// TIA Portal V17 export
// export: Created 2022-12-09T10:51:17.2356961Z, ExportSetting WithDefaults, DisplayName Totally Integrated Automation Portal, DisplayVersion V17 Update 5, DisplayName TIA Portal Openness, DisplayVersion V17 Update 5, DisplayName TIA Portal Version Control Interface, DisplayVersion V17, DisplayName Simotion SCOUT TIA, DisplayVersion 5.4.3.0, DisplayName SINAMICS Startdrive Advanced, DisplayVersion V17 SP1, DisplayName SINAMICS Startdrive G130, G150, S120, S150, SINAMICS MV, S210, DisplayVersion V17 SP1, DisplayName SINAMICS Startdrive G110M, G120, G120C, G120D, G120P, G115D, DisplayVersion V17 SP1, DisplayName STEP 7 Professional, DisplayVersion V17 Update 5, DisplayName STEP 7 Safety, DisplayVersion V17, DisplayName WinCC Advanced, DisplayVersion V17 Update 5
TYPE "UDT_OMAC_NamesConfiguration"
// stored: IsFailsafeCompliant false
   STRUCT
      unitModesNames : Array[0.."OMAC_LANGUAGES_UPPER_LIM", 0.."OMAC_MODES_UPPER_LIM"] of String[18];   // Names of unit modes [First index language, Second unit mode no] / 'UserModeXX'
      statesNames : Array[0.."OMAC_LANGUAGES_UPPER_LIM", 0.."OMAC_STATES_UPPER_LIM"] of String[16];   // Names of states [First index language, Second state no] / Names of states for [First index language, Second state no]
   END_STRUCT;
   // unitModesNames[0,0] := 'Invalid';
   // unitModesNames[0,1] := 'Production';
   // unitModesNames[0,2] := 'Maintenance';
   // unitModesNames[0,3] := 'Manual';
   // unitModesNames[0,4] := 'Change over';
   // unitModesNames[0,5] := 'Clean';
   // unitModesNames[0,6] := 'Set up';
   // unitModesNames[0,7] := 'Empty out';
   // unitModesNames[0,8] := 'OEM specific';
   // unitModesNames[0,9] := 'Spare';
   // unitModesNames[0,10] := 'User Mode 01';
   // unitModesNames[0,11] := 'User Mode 02';
   // unitModesNames[0,12] := 'User Mode 03';
   // unitModesNames[0,13] := 'User Mode 04';
   // unitModesNames[0,14] := 'User Mode 05';
   // unitModesNames[1,0] := 'Invalid';
   // unitModesNames[1,1] := 'Production';
   // unitModesNames[1,2] := 'Maintenance';
   // unitModesNames[1,3] := 'Manual';
   // unitModesNames[1,4] := 'Change over';
   // unitModesNames[1,5] := 'Clean';
   // unitModesNames[1,6] := 'Set up';
   // unitModesNames[1,7] := 'Empty out';
   // unitModesNames[1,8] := 'OEM specific';
   // unitModesNames[1,9] := 'Spare';
   // unitModesNames[1,10] := 'User Mode 01';
   // unitModesNames[1,11] := 'User Mode 02';
   // unitModesNames[1,12] := 'User Mode 03';
   // unitModesNames[1,13] := 'User Mode 04';
   // unitModesNames[1,14] := 'User Mode 05';
   // statesNames[0,0] := 'Undefined';
   // statesNames[0,1] := 'Clearing';
   // statesNames[0,2] := 'Stopped';
   // statesNames[0,3] := 'Starting';
   // statesNames[0,4] := 'Idle';
   // statesNames[0,5] := 'Suspended';
   // statesNames[0,6] := 'Execute';
   // statesNames[0,7] := 'Stopping';
   // statesNames[0,8] := 'Aborting';
   // statesNames[0,9] := 'Aborted';
   // statesNames[0,10] := 'Holding';
   // statesNames[0,11] := 'Held';
   // statesNames[0,12] := 'UnHolding';
   // statesNames[0,13] := 'Suspending';
   // statesNames[0,14] := 'UnSuspending';
   // statesNames[0,15] := 'Resetting';
   // statesNames[0,16] := 'Completing';
   // statesNames[0,17] := 'Complete';
   // statesNames[1,0] := 'Undefiniert';
   // statesNames[1,1] := 'Clearing';
   // statesNames[1,2] := 'Stopped';
   // statesNames[1,3] := 'Starting';
   // statesNames[1,4] := 'Idle';
   // statesNames[1,5] := 'Suspended';
   // statesNames[1,6] := 'Execute';
   // statesNames[1,7] := 'Stopping';
   // statesNames[1,8] := 'Aborting';
   // statesNames[1,9] := 'Aborted';
   // statesNames[1,10] := 'Holding';
   // statesNames[1,11] := 'Held';
   // statesNames[1,12] := 'UnHolding';
   // statesNames[1,13] := 'Suspending';
   // statesNames[1,14] := 'UnSuspending';
   // statesNames[1,15] := 'Resetting';
   // statesNames[1,16] := 'Completing';
   // statesNames[1,17] := 'Complete';
END_TYPE
